PROGRAM prgE9
VAR
	FB_Read_MB :FB_ModBus_100Registers_FC3;
	m_Enable: BOOL;
	str_IP: STRING(15):= '192.168.8.3';
	word_Adress: WORD;
	usint_Quantity: USINT;
	byte_slaveID: BYTE;
	
	lr_Bitumentank_1_Freq 			: LREAL;		//{#lynus.ag#()}
	lr_Bitumentank_1_L1N 			: LREAL;		//{#lynus.ag#()}
	lr_Bitumentank_1_L2N 			: LREAL;		//{#lynus.ag#()}
	lr_Bitumentank_1_L3N 			: LREAL;		//{#lynus.ag#()}
	lr_Bitumentank_1_L1L2 			: LREAL;		//{#lynus.ag#()}
	lr_Bitumentank_1_L2L3 			: LREAL;		//{#lynus.ag#()}
	lr_Bitumentank_1_L3L1 			: LREAL;		//{#lynus.ag#()}
	lr_Bitumentank_1_I1 			: LREAL;		//{#lynus.ag#()}
	lr_Bitumentank_1_I2 			: LREAL;		//{#lynus.ag#()}
	lr_Bitumentank_1_I3 			: LREAL;		//{#lynus.ag#()}
	lr_Bitumentank_1_N 				: LREAL;		//{#lynus.ag#()}
	lr_Bitumentank_1_S 				: LREAL;		//{#lynus.ag#()}
	lr_Bitumentank_1_P 				: LREAL;		//{#lynus.ag#()}
	lr_Bitumentank_1_Q 				: LREAL;		//{#lynus.ag#()}
	lr_Bitumentank_1_PF 			: LREAL;		//{#lynus.ag#()}
	
	lr_Bitumentank_2_Freq 			: LREAL;		//{#lynus.ag#()}
	lr_Bitumentank_2_L1N 			: LREAL;		//{#lynus.ag#()}
	lr_Bitumentank_2_L2N 			: LREAL;		//{#lynus.ag#()}
	lr_Bitumentank_2_L3N 			: LREAL;		//{#lynus.ag#()}
	lr_Bitumentank_2_L1L2 			: LREAL;		//{#lynus.ag#()}
	lr_Bitumentank_2_L2L3 			: LREAL;		//{#lynus.ag#()}
	lr_Bitumentank_2_L3L1 			: LREAL;		//{#lynus.ag#()}
	lr_Bitumentank_2_I1 			: LREAL;		//{#lynus.ag#()}
	lr_Bitumentank_2_I2 			: LREAL;		//{#lynus.ag#()}
	lr_Bitumentank_2_I3 			: LREAL;		//{#lynus.ag#()}
	lr_Bitumentank_2_N 				: LREAL;		//{#lynus.ag#()}
	lr_Bitumentank_2_S 				: LREAL;		//{#lynus.ag#()}
	lr_Bitumentank_2_P 				: LREAL;		//{#lynus.ag#()}
	lr_Bitumentank_2_Q 				: LREAL;		//{#lynus.ag#()}
	lr_Bitumentank_2_PF 			: LREAL;		//{#lynus.ag#()}
	
	lr_Bitumentank_3_Freq 			: LREAL;		//{#lynus.ag#()}
	lr_Bitumentank_3_L1N 			: LREAL;		//{#lynus.ag#()}
	lr_Bitumentank_3_L2N 			: LREAL;		//{#lynus.ag#()}
	lr_Bitumentank_3_L3N 			: LREAL;		//{#lynus.ag#()}
	lr_Bitumentank_3_L1L2 			: LREAL;		//{#lynus.ag#()}
	lr_Bitumentank_3_L2L3 			: LREAL;		//{#lynus.ag#()}
	lr_Bitumentank_3_L3L1 			: LREAL;		//{#lynus.ag#()}
	lr_Bitumentank_3_I1 			: LREAL;		//{#lynus.ag#()}
	lr_Bitumentank_3_I2 			: LREAL;		//{#lynus.ag#()}
	lr_Bitumentank_3_I3 			: LREAL;		//{#lynus.ag#()}
	lr_Bitumentank_3_N 				: LREAL;		//{#lynus.ag#()}
	lr_Bitumentank_3_S 				: LREAL;		//{#lynus.ag#()}
	lr_Bitumentank_3_P 				: LREAL;		//{#lynus.ag#()}
	lr_Bitumentank_3_Q 				: LREAL;		//{#lynus.ag#()}
	lr_Bitumentank_3_PF 			: LREAL;		//{#lynus.ag#()}
	
	lr_Bitumentank_4_Freq 			: LREAL;		//{#lynus.ag#()}
	lr_Bitumentank_4_L1N 			: LREAL;		//{#lynus.ag#()}
	lr_Bitumentank_4_L2N 			: LREAL;		//{#lynus.ag#()}
	lr_Bitumentank_4_L3N 			: LREAL;		//{#lynus.ag#()}
	lr_Bitumentank_4_L1L2 			: LREAL;		//{#lynus.ag#()}
	lr_Bitumentank_4_L2L3 			: LREAL;		//{#lynus.ag#()}
	lr_Bitumentank_4_L3L1 			: LREAL;		//{#lynus.ag#()}
	lr_Bitumentank_4_I1 			: LREAL;		//{#lynus.ag#()}
	lr_Bitumentank_4_I2 			: LREAL;		//{#lynus.ag#()}
	lr_Bitumentank_4_I3 			: LREAL;		//{#lynus.ag#()}
	lr_Bitumentank_4_N 				: LREAL;		//{#lynus.ag#()}
	lr_Bitumentank_4_S 				: LREAL;		//{#lynus.ag#()}
	lr_Bitumentank_4_P 				: LREAL;		//{#lynus.ag#()}
	lr_Bitumentank_4_Q 				: LREAL;		//{#lynus.ag#()}
	lr_Bitumentank_4_PF 			: LREAL;		//{#lynus.ag#()}
	
	lr_Bitumenfuellpumpe_1_Freq 	: LREAL;		//{#lynus.ag#()}
	lr_Bitumenfuellpumpe_1_L1N 		: LREAL;		//{#lynus.ag#()}
	lr_Bitumenfuellpumpe_1_L2N 		: LREAL;		//{#lynus.ag#()}
	lr_Bitumenfuellpumpe_1_L3N 		: LREAL;		//{#lynus.ag#()}
	lr_Bitumenfuellpumpe_1_L1L2 	: LREAL;		//{#lynus.ag#()}
	lr_Bitumenfuellpumpe_1_L2L3 	: LREAL;		//{#lynus.ag#()}
	lr_Bitumenfuellpumpe_1_L3L1		: LREAL;		//{#lynus.ag#()}
	lr_Bitumenfuellpumpe_1_I1 		: LREAL;		//{#lynus.ag#()}
	lr_Bitumenfuellpumpe_1_I2 		: LREAL;		//{#lynus.ag#()}
	lr_Bitumenfuellpumpe_1_I3 		: LREAL;		//{#lynus.ag#()}
	lr_Bitumenfuellpumpe_1_N 		: LREAL;		//{#lynus.ag#()}
	lr_Bitumenfuellpumpe_1_S 		: LREAL;		//{#lynus.ag#()}
	lr_Bitumenfuellpumpe_1_P 		: LREAL;		//{#lynus.ag#()}
	lr_Bitumenfuellpumpe_1_Q 		: LREAL;		//{#lynus.ag#()}
	lr_Bitumenfuellpumpe_1_PF 		: LREAL;		//{#lynus.ag#()}

	lr_Dosierpumpe_1_Freq 			: LREAL;		//{#lynus.ag#()}
	lr_Dosierpumpe_1_L1N 			: LREAL;		//{#lynus.ag#()}
	lr_Dosierpumpe_1_L2N 			: LREAL;		//{#lynus.ag#()}
	lr_Dosierpumpe_1_L3N 			: LREAL;		//{#lynus.ag#()}
	lr_Dosierpumpe_1_L1L2 			: LREAL;		//{#lynus.ag#()}
	lr_Dosierpumpe_1_L2L3 			: LREAL;		//{#lynus.ag#()}
	lr_Dosierpumpe_1_L3L1 			: LREAL;		//{#lynus.ag#()}
	lr_Dosierpumpe_1_I1 			: LREAL;		//{#lynus.ag#()}
	lr_Dosierpumpe_1_I2 			: LREAL;		//{#lynus.ag#()}
	lr_Dosierpumpe_1_I3 			: LREAL;		//{#lynus.ag#()}
	lr_Dosierpumpe_1_N 				: LREAL;		//{#lynus.ag#()}
	lr_Dosierpumpe_1_S 				: LREAL;		//{#lynus.ag#()}
	lr_Dosierpumpe_1_P 				: LREAL;		//{#lynus.ag#()}
	lr_Dosierpumpe_1_Q 				: LREAL;		//{#lynus.ag#()}
	lr_Dosierpumpe_1_PF 			: LREAL;		//{#lynus.ag#()}

	lr_Dosierpumpe_2_Freq 			: LREAL;		//{#lynus.ag#()}
	lr_Dosierpumpe_2_L1N 			: LREAL;		//{#lynus.ag#()}
	lr_Dosierpumpe_2_L2N 			: LREAL;		//{#lynus.ag#()}
	lr_Dosierpumpe_2_L3N 			: LREAL;		//{#lynus.ag#()}
	lr_Dosierpumpe_2_L1L2 			: LREAL;		//{#lynus.ag#()}
	lr_Dosierpumpe_2_L2L3 			: LREAL;		//{#lynus.ag#()}
	lr_Dosierpumpe_2_L3L1 			: LREAL;		//{#lynus.ag#()}
	lr_Dosierpumpe_2_I1 			: LREAL;		//{#lynus.ag#()}
	lr_Dosierpumpe_2_I2 			: LREAL;		//{#lynus.ag#()}
	lr_Dosierpumpe_2_I3 			: LREAL;		//{#lynus.ag#()}
	lr_Dosierpumpe_2_N 				: LREAL;		//{#lynus.ag#()}
	lr_Dosierpumpe_2_S 				: LREAL;		//{#lynus.ag#()}
	lr_Dosierpumpe_2_P 				: LREAL;		//{#lynus.ag#()}
	lr_Dosierpumpe_2_Q 				: LREAL;		//{#lynus.ag#()}
	lr_Dosierpumpe_2_PF 			: LREAL;		//{#lynus.ag#()}
	
	m_Bitumenfuellpumpe_1	 		: BOOL;			//{#lynus.ag#()}
	
	FB_Read_Socomec_I61 	: FB_Socomec_I61;
	FB_Read_Socomec_I31 	: FB_Socomec_I31;
	FB_Read_Socomec_IO10	: FB_Socomec_IO10;
	i_State_ModbusCall: INT;				
	ton_TimeOutState: ton;
	tof_TimeOut_Active: tof;
	i_State_ModbusCall_old: INT;
	int_errorCount: INT;
	m_TimeOutActive: BOOL;					//{#lynus.ag#()}
	i_State_ErrorActive: INT;				//{#lynus.ag#()}
END_VAR

CASE i_State_ModbusCall OF
	0: 	// wait state
		i_State_ModbusCall := 10;
	
	10:	// first Modbus Poll Call
		FB_Read_Socomec_I61.m_Start := TRUE;
		FB_Read_Socomec_I61.byte_slaveID := 26;
		FB_Read_Socomec_I61.w_Adress := 18442;
		i_State_ModbusCall := i_State_ModbusCall + 1;
	
	11: // wait for received data
		FB_Read_Socomec_I61.m_Start := FALSE;
		IF FB_Read_Socomec_I61.iStateModbusRead = 30 THEN
			lr_Bitumentank_4_Freq	:=		FB_Read_Socomec_I61.lr_Freq_Hz	;	
			lr_Bitumentank_4_L1N	:=		FB_Read_Socomec_I61.lr_L1N_V	;	
			lr_Bitumentank_4_L2N	:=		FB_Read_Socomec_I61.lr_L2N_V	;	
			lr_Bitumentank_4_L3N	:=		FB_Read_Socomec_I61.lr_L3N_V	;	
			lr_Bitumentank_4_L1L2	:=		FB_Read_Socomec_I61.lr_L1L2_V	;	
			lr_Bitumentank_4_L2L3	:=		FB_Read_Socomec_I61.lr_L2L3_V	;	
			lr_Bitumentank_4_L3L1	:=		FB_Read_Socomec_I61.lr_L3L1_V	;	
			lr_Bitumentank_4_I1		:=		FB_Read_Socomec_I61.lr_I1_A		;	
			lr_Bitumentank_4_I2		:=		FB_Read_Socomec_I61.lr_I2_A		;	
			lr_Bitumentank_4_I3		:=		FB_Read_Socomec_I61.lr_I3_A		;	
			lr_Bitumentank_4_N		:=		FB_Read_Socomec_I61.lr_N_A		;	
			lr_Bitumentank_4_P		:=		FB_Read_Socomec_I61.lr_P_kW		;	
			lr_Bitumentank_4_Q		:=		FB_Read_Socomec_I61.lr_Q_kVAr	;	
			lr_Bitumentank_4_S		:=		FB_Read_Socomec_I61.lr_S_kVA	;	
			lr_Bitumentank_4_PF		:=		FB_Read_Socomec_I61.lr_PF		;		
			
			i_State_ModbusCall := i_State_ModbusCall +1;
		END_IF            
		IF FB_Read_Socomec_I61.iStateModbusError = 300 OR ton_TimeOutState.Q THEN
			i_State_ModbusCall := i_State_ModbusCall +1;
		END_IF
	
	12: // wait for FB_Read_Socomec_I61 to be in state 0
		IF FB_Read_Socomec_I61.iStateModbusRead = 0 OR ton_TimeOutState.Q THEN
			i_State_ModbusCall := i_State_ModbusCall + 8;
		END_IF

	20:	// next Modbus Poll Call
		FB_Read_Socomec_I61.m_Start := TRUE;
		FB_Read_Socomec_I61.byte_slaveID := 27;
		FB_Read_Socomec_I61.w_Adress := 18442;
		i_State_ModbusCall := i_State_ModbusCall + 1;
	
	21: // wait for received data
		FB_Read_Socomec_I61.m_Start := FALSE;
		IF FB_Read_Socomec_I61.iStateModbusRead = 30 THEN
			lr_Dosierpumpe_1_Freq		:=		FB_Read_Socomec_I61.lr_Freq_Hz	;	
			lr_Dosierpumpe_1_L1N		:=		FB_Read_Socomec_I61.lr_L1N_V	;	
			lr_Dosierpumpe_1_L2N		:=		FB_Read_Socomec_I61.lr_L2N_V	;	
			lr_Dosierpumpe_1_L3N		:=		FB_Read_Socomec_I61.lr_L3N_V	;	
			lr_Dosierpumpe_1_L1L2		:=		FB_Read_Socomec_I61.lr_L1L2_V	;	
			lr_Dosierpumpe_1_L2L3		:=		FB_Read_Socomec_I61.lr_L2L3_V	;	
			lr_Dosierpumpe_1_L3L1		:=		FB_Read_Socomec_I61.lr_L3L1_V	;	
			lr_Dosierpumpe_1_I1			:=		FB_Read_Socomec_I61.lr_I1_A		;	
			lr_Dosierpumpe_1_I2			:=		FB_Read_Socomec_I61.lr_I2_A		;	
			lr_Dosierpumpe_1_I3			:=		FB_Read_Socomec_I61.lr_I3_A		;	
			lr_Dosierpumpe_1_N			:=		FB_Read_Socomec_I61.lr_N_A		;	
			lr_Dosierpumpe_1_P			:=		FB_Read_Socomec_I61.lr_P_kW		;	
			lr_Dosierpumpe_1_Q			:=		FB_Read_Socomec_I61.lr_Q_kVAr	;	
			lr_Dosierpumpe_1_S			:=		FB_Read_Socomec_I61.lr_S_kVA	;	
			lr_Dosierpumpe_1_PF			:=		FB_Read_Socomec_I61.lr_PF		;		
			
			i_State_ModbusCall := i_State_ModbusCall +1;
		END_IF            
		IF FB_Read_Socomec_I61.iStateModbusError = 300 OR ton_TimeOutState.Q THEN
			i_State_ModbusCall := i_State_ModbusCall +1;
		END_IF
	
	22: // wait for FB_Read_Socomec_I61 to be in state 0
		IF FB_Read_Socomec_I61.iStateModbusRead = 0 OR ton_TimeOutState.Q THEN
			i_State_ModbusCall := i_State_ModbusCall + 8;
		END_IF
	
	30:	// next Modbus Poll Call
		FB_Read_Socomec_I61.m_Start := TRUE;
		FB_Read_Socomec_I61.byte_slaveID := 26;
		FB_Read_Socomec_I61.w_Adress := 20490;
		i_State_ModbusCall := i_State_ModbusCall + 1;
	
	31: // wait for received data
		FB_Read_Socomec_I61.m_Start := FALSE;
		IF FB_Read_Socomec_I61.iStateModbusRead = 30 THEN
			lr_Bitumenfuellpumpe_1_Freq		:=		FB_Read_Socomec_I61.lr_Freq_Hz	;	
			lr_Bitumenfuellpumpe_1_L1N		:=		FB_Read_Socomec_I61.lr_L1N_V	;	
			lr_Bitumenfuellpumpe_1_L2N		:=		FB_Read_Socomec_I61.lr_L2N_V	;	
			lr_Bitumenfuellpumpe_1_L3N		:=		FB_Read_Socomec_I61.lr_L3N_V	;	
			lr_Bitumenfuellpumpe_1_L1L2		:=		FB_Read_Socomec_I61.lr_L1L2_V	;	
			lr_Bitumenfuellpumpe_1_L2L3		:=		FB_Read_Socomec_I61.lr_L2L3_V	;	
			lr_Bitumenfuellpumpe_1_L3L1		:=		FB_Read_Socomec_I61.lr_L3L1_V	;	
			lr_Bitumenfuellpumpe_1_I1		:=		FB_Read_Socomec_I61.lr_I1_A		;	
			lr_Bitumenfuellpumpe_1_I2		:=		FB_Read_Socomec_I61.lr_I2_A		;	
			lr_Bitumenfuellpumpe_1_I3		:=		FB_Read_Socomec_I61.lr_I3_A		;	
			lr_Bitumenfuellpumpe_1_N		:=		FB_Read_Socomec_I61.lr_N_A		;	
			lr_Bitumenfuellpumpe_1_P		:=		FB_Read_Socomec_I61.lr_P_kW		;	
			lr_Bitumenfuellpumpe_1_Q		:=		FB_Read_Socomec_I61.lr_Q_kVAr	;	
			lr_Bitumenfuellpumpe_1_S		:=		FB_Read_Socomec_I61.lr_S_kVA	;	
			lr_Bitumenfuellpumpe_1_PF		:=		FB_Read_Socomec_I61.lr_PF		;		
			
			i_State_ModbusCall := i_State_ModbusCall +1;
		END_IF            
		IF FB_Read_Socomec_I61.iStateModbusError = 300 OR ton_TimeOutState.Q THEN
			i_State_ModbusCall := i_State_ModbusCall +1;
		END_IF
	
	32: // wait for FB_Read_Socomec_I61 to be in state 0
		IF FB_Read_Socomec_I61.iStateModbusRead = 0 OR ton_TimeOutState.Q THEN
			i_State_ModbusCall := i_State_ModbusCall + 8;
		END_IF
	
	40:	// next Modbus Poll Call
		FB_Read_Socomec_I61.m_Start := TRUE;
		FB_Read_Socomec_I61.byte_slaveID := 27;
		FB_Read_Socomec_I61.w_Adress := 20490;
		i_State_ModbusCall := i_State_ModbusCall + 1;
	
	41: // wait for received data
		FB_Read_Socomec_I61.m_Start := FALSE;
		IF FB_Read_Socomec_I61.iStateModbusRead = 30 THEN
			lr_Dosierpumpe_2_Freq	:=		FB_Read_Socomec_I61.lr_Freq_Hz	;	
			lr_Dosierpumpe_2_L1N	:=		FB_Read_Socomec_I61.lr_L1N_V	;	
			lr_Dosierpumpe_2_L2N	:=		FB_Read_Socomec_I61.lr_L2N_V	;	
			lr_Dosierpumpe_2_L3N	:=		FB_Read_Socomec_I61.lr_L3N_V	;	
			lr_Dosierpumpe_2_L1L2	:=		FB_Read_Socomec_I61.lr_L1L2_V	;	
			lr_Dosierpumpe_2_L2L3	:=		FB_Read_Socomec_I61.lr_L2L3_V	;	
			lr_Dosierpumpe_2_L3L1	:=		FB_Read_Socomec_I61.lr_L3L1_V	;	
			lr_Dosierpumpe_2_I1		:=		FB_Read_Socomec_I61.lr_I1_A		;	
			lr_Dosierpumpe_2_I2		:=		FB_Read_Socomec_I61.lr_I2_A		;	
			lr_Dosierpumpe_2_I3		:=		FB_Read_Socomec_I61.lr_I3_A		;	
			lr_Dosierpumpe_2_N		:=		FB_Read_Socomec_I61.lr_N_A		;	
			lr_Dosierpumpe_2_P		:=		FB_Read_Socomec_I61.lr_P_kW		;	
			lr_Dosierpumpe_2_Q		:=		FB_Read_Socomec_I61.lr_Q_kVAr	;	
			lr_Dosierpumpe_2_S		:=		FB_Read_Socomec_I61.lr_S_kVA	;	
			lr_Dosierpumpe_2_PF		:=		FB_Read_Socomec_I61.lr_PF		;		
			
			i_State_ModbusCall := i_State_ModbusCall +1;
		END_IF            
		IF FB_Read_Socomec_I61.iStateModbusError = 300 OR ton_TimeOutState.Q THEN
			i_State_ModbusCall := i_State_ModbusCall +1;
		END_IF
	
	42: // wait for FB_Read_Socomec_I61 to be in state 0
		IF FB_Read_Socomec_I61.iStateModbusRead = 0 OR ton_TimeOutState.Q THEN
			i_State_ModbusCall := i_State_ModbusCall + 8;
		END_IF

	50:	// next Modbus Poll Call		first IO10 call
		FB_Read_Socomec_IO10.m_Start := TRUE;
		FB_Read_Socomec_IO10.byte_slaveID := 28;
		FB_Read_Socomec_IO10.w_Adress := 11520;
		i_State_ModbusCall := i_State_ModbusCall + 1;
	
	51: // wait for received data
		FB_Read_Socomec_IO10.m_Start := FALSE;
		IF FB_Read_Socomec_IO10.iStateModbusRead = 30 THEN
			m_Bitumenfuellpumpe_1 := FB_Read_Socomec_IO10.m_Input_Active;		
				
			i_State_ModbusCall := i_State_ModbusCall +1;
		END_IF            
		IF FB_Read_Socomec_IO10.iStateModbusError = 300 OR ton_TimeOutState.Q THEN
			i_State_ModbusCall := i_State_ModbusCall +1;
		END_IF
	
	52: // wait for FB_Read_Socomec_IO10 to be in state 0
		IF FB_Read_Socomec_IO10.iStateModbusRead = 0 OR ton_TimeOutState.Q THEN
			i_State_ModbusCall := i_State_ModbusCall + 8;
		END_IF
		
	60:	// next Modbus Poll Call
		FB_Read_Socomec_I31.m_Start := TRUE;
		FB_Read_Socomec_I31.byte_slaveID := 23;
		FB_Read_Socomec_I31.w_Adress := 18442;
		i_State_ModbusCall := i_State_ModbusCall + 1;
	
	61: // wait for received data
		FB_Read_Socomec_I31.m_Start := FALSE;
		IF FB_Read_Socomec_I31.iStateModbusRead = 30 THEN
			lr_Bitumentank_1_Freq	:=		FB_Read_Socomec_I31.lr_Freq_Hz	;	
			lr_Bitumentank_1_L1N	:=		FB_Read_Socomec_I31.lr_L1N_V	;	
			lr_Bitumentank_1_L2N	:=		FB_Read_Socomec_I31.lr_L2N_V	;	
			lr_Bitumentank_1_L3N	:=		FB_Read_Socomec_I31.lr_L3N_V	;	
			lr_Bitumentank_1_L1L2	:=		FB_Read_Socomec_I31.lr_L1L2_V	;	
			lr_Bitumentank_1_L2L3	:=		FB_Read_Socomec_I31.lr_L2L3_V	;	
			lr_Bitumentank_1_L3L1	:=		FB_Read_Socomec_I31.lr_L3L1_V	;	
			lr_Bitumentank_1_I1		:=		FB_Read_Socomec_I31.lr_I1_A		;	
			lr_Bitumentank_1_I2		:=		FB_Read_Socomec_I31.lr_I2_A		;	
			lr_Bitumentank_1_I3		:=		FB_Read_Socomec_I31.lr_I3_A		;	
			lr_Bitumentank_1_N		:=		FB_Read_Socomec_I31.lr_N_A		;	
			lr_Bitumentank_1_P		:=		FB_Read_Socomec_I31.lr_P_kW		;	
			lr_Bitumentank_1_Q		:=		FB_Read_Socomec_I31.lr_Q_kVAr	;	
			lr_Bitumentank_1_S		:=		FB_Read_Socomec_I31.lr_S_kVA	;	
			lr_Bitumentank_1_PF		:=		FB_Read_Socomec_I31.lr_PF		;		
			
			i_State_ModbusCall := i_State_ModbusCall +1;
		END_IF            
		IF FB_Read_Socomec_I31.iStateModbusError = 300 OR ton_TimeOutState.Q THEN
			i_State_ModbusCall := i_State_ModbusCall +1;
		END_IF
	
	62: // wait for FB_Read_Socomec_I31 to be in state 0
		IF FB_Read_Socomec_I31.iStateModbusRead = 0 OR ton_TimeOutState.Q THEN
			i_State_ModbusCall := i_State_ModbusCall + 8;
		END_IF
		
	70:	// next Modbus Poll Call
		FB_Read_Socomec_I31.m_Start := TRUE;
		FB_Read_Socomec_I31.byte_slaveID := 24;
		FB_Read_Socomec_I31.w_Adress := 18442;
		i_State_ModbusCall := i_State_ModbusCall + 1;
	
	71: // wait for received data
		FB_Read_Socomec_I31.m_Start := FALSE;
		IF FB_Read_Socomec_I31.iStateModbusRead = 30 THEN
			lr_Bitumentank_2_Freq	:=		FB_Read_Socomec_I31.lr_Freq_Hz	;	
			lr_Bitumentank_2_L1N	:=		FB_Read_Socomec_I31.lr_L1N_V	;	
			lr_Bitumentank_2_L2N	:=		FB_Read_Socomec_I31.lr_L2N_V	;	
			lr_Bitumentank_2_L3N	:=		FB_Read_Socomec_I31.lr_L3N_V	;	
			lr_Bitumentank_2_L1L2	:=		FB_Read_Socomec_I31.lr_L1L2_V	;	
			lr_Bitumentank_2_L2L3	:=		FB_Read_Socomec_I31.lr_L2L3_V	;	
			lr_Bitumentank_2_L3L1	:=		FB_Read_Socomec_I31.lr_L3L1_V	;	
			lr_Bitumentank_2_I1		:=		FB_Read_Socomec_I31.lr_I1_A		;	
			lr_Bitumentank_2_I2		:=		FB_Read_Socomec_I31.lr_I2_A		;	
			lr_Bitumentank_2_I3		:=		FB_Read_Socomec_I31.lr_I3_A		;	
			lr_Bitumentank_2_N		:=		FB_Read_Socomec_I31.lr_N_A		;	
			lr_Bitumentank_2_P		:=		FB_Read_Socomec_I31.lr_P_kW		;	
			lr_Bitumentank_2_Q		:=		FB_Read_Socomec_I31.lr_Q_kVAr	;	
			lr_Bitumentank_2_S		:=		FB_Read_Socomec_I31.lr_S_kVA	;	
			lr_Bitumentank_2_PF		:=		FB_Read_Socomec_I31.lr_PF		;		
			
			i_State_ModbusCall := i_State_ModbusCall +1;
		END_IF            
		IF FB_Read_Socomec_I31.iStateModbusError = 300 OR ton_TimeOutState.Q THEN
			i_State_ModbusCall := i_State_ModbusCall +1;
		END_IF
	
	72: // wait for FB_Read_Socomec_I31 to be in state 0
		IF FB_Read_Socomec_I31.iStateModbusRead = 0 OR ton_TimeOutState.Q THEN
			i_State_ModbusCall := i_State_ModbusCall + 8;
		END_IF
		
	80:	// next Modbus Poll Call
		FB_Read_Socomec_I31.m_Start := TRUE;
		FB_Read_Socomec_I31.byte_slaveID := 25;
		FB_Read_Socomec_I31.w_Adress := 18442;
		i_State_ModbusCall := i_State_ModbusCall + 1;
	
	81: // wait for received data
		FB_Read_Socomec_I31.m_Start := FALSE;
		IF FB_Read_Socomec_I31.iStateModbusRead = 30 THEN
			lr_Bitumentank_3_Freq	:=		FB_Read_Socomec_I31.lr_Freq_Hz	;	
			lr_Bitumentank_3_L1N	:=		FB_Read_Socomec_I31.lr_L1N_V	;	
			lr_Bitumentank_3_L2N	:=		FB_Read_Socomec_I31.lr_L2N_V	;	
			lr_Bitumentank_3_L3N	:=		FB_Read_Socomec_I31.lr_L3N_V	;	
			lr_Bitumentank_3_L1L2	:=		FB_Read_Socomec_I31.lr_L1L2_V	;	
			lr_Bitumentank_3_L2L3	:=		FB_Read_Socomec_I31.lr_L2L3_V	;	
			lr_Bitumentank_3_L3L1	:=		FB_Read_Socomec_I31.lr_L3L1_V	;	
			lr_Bitumentank_3_I1		:=		FB_Read_Socomec_I31.lr_I1_A		;	
			lr_Bitumentank_3_I2		:=		FB_Read_Socomec_I31.lr_I2_A		;	
			lr_Bitumentank_3_I3		:=		FB_Read_Socomec_I31.lr_I3_A		;	
			lr_Bitumentank_3_N		:=		FB_Read_Socomec_I31.lr_N_A		;	
			lr_Bitumentank_3_P		:=		FB_Read_Socomec_I31.lr_P_kW		;	
			lr_Bitumentank_3_Q		:=		FB_Read_Socomec_I31.lr_Q_kVAr	;	
			lr_Bitumentank_3_S		:=		FB_Read_Socomec_I31.lr_S_kVA	;	
			lr_Bitumentank_3_PF		:=		FB_Read_Socomec_I31.lr_PF		;		
			
			i_State_ModbusCall := i_State_ModbusCall +1;
		END_IF            
		IF FB_Read_Socomec_I31.iStateModbusError = 300 OR ton_TimeOutState.Q THEN
			i_State_ModbusCall := i_State_ModbusCall +1;
		END_IF
	
	82: // wait for FB_Read_Socomec_I31 to be in state 0
		IF FB_Read_Socomec_I31.iStateModbusRead = 0 OR ton_TimeOutState.Q THEN
			i_State_ModbusCall := i_State_ModbusCall + 8;
		END_IF
		
	90: 
		i_State_ModbusCall := 0;
		
END_CASE

ton_TimeOutState(	IN:= i_State_ModbusCall = i_State_ModbusCall_old, 
					PT:= T#30S, 
					Q=> , 
					ET=> );

i_State_ModbusCall_old := i_State_ModbusCall; 

IF ton_TimeOutState.Q THEN
//	i_State_ModbusCall := 0;
	int_errorCount := int_errorCount  + 1; 
END_IF


tof_TimeOut_Active(	IN:= ton_TimeOutState.Q, 
					PT:=	T#5S , 
					Q=> m_TimeOutActive, 
					ET=> );
IF tof_TimeOut_Active.Q THEN
	 i_State_ErrorActive := i_State_ModbusCall; 
END_IF


FB_Read_Socomec_I61(
	m_Start:= , 
	str_IPAdress:= str_IP , 
	w_Adress:= , 
	uint_port:= , 
	byte_slaveID:= , 
	m_PollSuccessful=> , 
	lr_Freq_Hz=> , 
	lr_L1N_V=> , 
	lr_L2N_V=> , 
	lr_L3N_V=> , 
	lr_L1L2_V=> , 
	lr_L2L3_V=> , 
	lr_L3L1_V=> , 
	lr_I1_A=> , 
	lr_I2_A=> , 
	lr_I3_A=> , 
	lr_N_A=> , 
	lr_P_kW=> , 
	lr_Q_kVAr=> , 
	lr_S_kVA=> , 
	lr_PF=> , 
	udint_Error_ID=> );
	
FB_Read_Socomec_I31(
	m_Start:= , 
	str_IPAdress:= str_IP , 
	w_Adress:= , 
	uint_port:= , 
	byte_slaveID:= , 
	m_PollSuccessful=> , 
	lr_Freq_Hz=> , 
	lr_L1N_V=> , 
	lr_L2N_V=> , 
	lr_L3N_V=> , 
	lr_L1L2_V=> , 
	lr_L2L3_V=> , 
	lr_L3L1_V=> , 
	lr_I1_A=> , 
	lr_I2_A=> , 
	lr_I3_A=> , 
	lr_N_A=> , 
	lr_P_kW=> , 
	lr_Q_kVAr=> , 
	lr_S_kVA=> , 
	lr_PF=> , 
	udint_Error_ID=> );

FB_Read_Socomec_IO10(
	m_Start:= , 
	str_IPAdress:= str_IP , 
	w_Adress:= , 
	uint_port:= , 
	byte_slaveID:= , 
	m_PollSuccessful=> , 
	m_Input_Active=> , 
	udint_Error_ID=> );	

FB_Read_MB(
	m_Enable:= m_Enable, 
	str_IPAdress:= str_IP,
	w_Adress:= word_Adress, 
	usint_Quantity:= usint_Quantity, 
	byte_slaveID:=byte_slaveID,
	uint_port := ,
	m_PollSuccessful=> , 
	w_Array_Received=> , 
	udint_Error_ID=> );

END_PROGRAM

(* stored: Version 1.1.0.1, ProductVersion 3.1.4024.12
   POU prgE9: Id {ded2e15b-e0fe-49a5-a52a-37de718b51d3}, SpecialFunc None *)
